(* PLC project Unnamed, Unknown Unnamed 1 *)
(* stored: creationDateTime 2025-09-07T23:21:20, modificationDateTime 2025-09-08T13:14:57 *)

PROGRAM program0
  VAR
    TON3 : TON;
    TON0 : TON;
    TON4 : DINT;
    TON1 : TON;
    INPUT_1 : BOOL;
    INPUT_2 : BOOL;
    INPUT_3 : BOOL;
    INPUT_4 : BOOL;
    INPUT_5 : BOOL;
    INPUT_6 : BOOL;
    INPUT_7 : BOOL;
    INPUT_8 : BOOL;
    INPUT_9 : BOOL;
    Switch : BOOL;
    Run : BOOL;
    manual_switch : BOOL;
    start_A : BOOL;
    strat_B : BOOL;
    INPUT_15 : BOOL;
    TON2 : TON;
    SR0 : SR;
    OUTOUT_1 : BOOL;
    Output_2 : BOOL;
    Indicator_Light : BOOL;
    OUTOUT_4 : BOOL;
    OUTOUT_5 : BOOL;
    OUTOUT_6 : BOOL;
  END_VAR

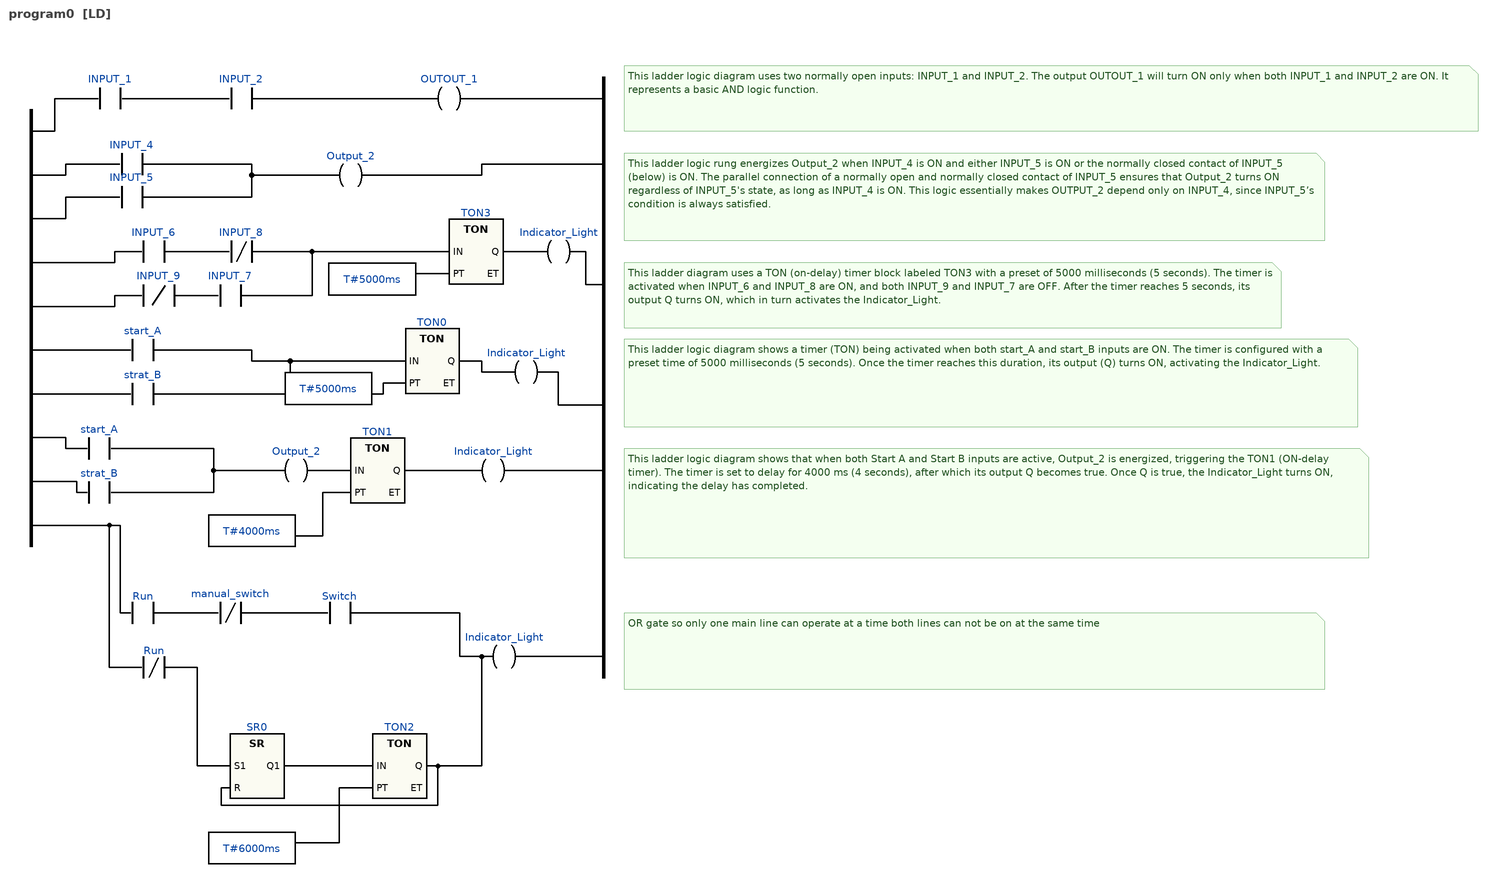
(* LD diagram, written out as Structured Text *)
(* This ladder logic diagram uses two normally open inputs: INPUT_1 and INPUT_2. The output OUTOUT_1 will turn ON only when both INPUT_1 and INPUT_2 are ON. It represents a basic AND logic function. *)
OUTOUT_1 := INPUT_1 AND INPUT_2;
(* This ladder logic rung energizes Output_2 when INPUT_4 is ON and either INPUT_5 is ON or the normally closed contact of INPUT_5 (below) is ON. The parallel connection of a normally open and normally closed contact of INPUT_5 ensures that Output_2 turns ON regardless of INPUT_5's state, as long as INPUT_4 is ON. This logic essentially makes OUTPUT_2 depend only on INPUT_4, since INPUT_5’s condition is always satisfied. *)
Output_2 := INPUT_4 OR INPUT_5;
TON3(IN := NOT INPUT_9 AND INPUT_7 OR INPUT_6 AND NOT INPUT_8, PT := T#5000ms);
Indicator_Light := TON3.Q;
(* This ladder diagram uses a TON (on-delay) timer block labeled TON3 with a preset of 5000 milliseconds (5 seconds). The timer is activated when INPUT_6 and INPUT_8 are ON, and both INPUT_9 and INPUT_7 are OFF. After the timer reaches 5 seconds, its output Q turns ON, which in turn activates the Indicator_Light. *)
(* This ladder logic diagram shows a timer (TON) being activated when both start_A and start_B inputs are ON. The timer is configured with a preset time of 5000 milliseconds (5 seconds). Once the timer reaches this duration, its output (Q) turns ON, activating the Indicator_Light. *)
TON0(IN := start_A OR strat_B, PT := T#5000ms);
Indicator_Light := TON0.Q;
(* This ladder logic diagram shows that when both Start A and Start B inputs are active, Output_2 is energized, triggering the TON1 (ON-delay timer). The timer is set to delay for 4000 ms (4 seconds), after which its output Q becomes true. Once Q is true, the Indicator_Light turns ON, indicating the delay has completed. *)
TON1(IN := start_A OR strat_B, PT := T#4000ms);
Indicator_Light := TON1.Q;
Output_2 := start_A OR strat_B;
(* OR gate so only one main line can operate at a time both lines can not be on at the same time *)
SR0(S1 := NOT Run, R := TON2.Q);
TON2(IN := SR0.Q1, PT := T#6000ms);
Indicator_Light := Run AND NOT manual_switch AND Switch OR TON2.Q;
END_PROGRAM

CONFIGURATION Config0
  RESOURCE Res0 ON PLC
    TASK task0(INTERVAL := T#20ms, PRIORITY := 0);
    PROGRAM instance0 WITH task0 : program0;
  END_RESOURCE
END_CONFIGURATION
